// TIA Portal V18 export
// export: Created 2025-12-01T17:52:58.631124Z, ExportSetting None, DisplayName Totally Integrated Automation Portal, DisplayVersion V18 Update 5, DisplayName TIA Portal Openness, DisplayVersion V18 Update 5, DisplayName TIA Portal Teamcenter Gateway, DisplayVersion V18, DisplayName TIA Portal Version Control Interface, DisplayVersion V18, DisplayName STEP 7 Professional, DisplayVersion V18 Update 5, DisplayName STEP 7 Safety, DisplayVersion V18, DisplayName WinCC Professional, DisplayVersion V18 Update 5
Screen "222 Scanner_806A1"  1280x800, Number=222, Template=02ManualUnit1
  ScreenLayer "Layer_0"
    FaceplateInstance "RCS_fpKeyenceSR1000_TP1200_1" at 10,129 size 1134x421  FaceplateTypeName=KeyenceSR1000@$@03_FacePlate@$@RCS_fpKeyenceSR1000_TP1200 V 0.0.6
      InterfacePropertyText "文本"  Text="806A1_MagentScan"
      Property := KeyenceSR1000Ctrl_806A1DB_sHMI
    Button "btnMenu4" at 384,725 size 128x75  TextOff="读码器_806A1 / Code reader 806A1", TextOn="读码器_806A1 / Code reader 806A1"
      on Click: ActivateScreen(Screen name := , Object number := 0)
    Button "btnMenu5" at 512,725 size 128x75  TextOff="气缸_B2 / Cylinder _B2", TextOn="气缸_B2 / Cylinder _B2"
      on Click: ActivateScreen(Screen name := 226_Cylinder_B2, Object number := 0)
    Button "btnMenu6" at 640,725 size 128x75  TextOff="压机_375A1 / Press_375A1", TextOn="压机_375A1 / Press_375A1"
      on Click: ActivateScreen(Screen name := 227 Kistler_375A1, Object number := 0)
    Button "btnMenu6_1" at 768,725 size 128x75
    Button "按钮_1" at 128,725 size 128x75  PictureOff=向右箭头_0, TextOff="气缸_B1 / Cylinder _B1", TextOn="气缸_B1 / Cylinder _B1"
      on Click: ActivateScreen(Screen name := 220_Cylinder_B1, Object number := 0)
    Button "btnMenu4_1" at 256,725 size 128x75  TextOff="压机_372A1 / Press_372A1", TextOn="压机_372A1 / Press_372A1"
      on Click: ActivateScreen(Screen name := 221 Kistler__372A1, Object number := 0)
    Button "btnMenu7" at 896,725 size 128x75
    Button "btnMenu7_1" at 1024,725 size 128x75
